// TIA Portal V19 export
ORGANIZATION_BLOCK "Main"   // OB1, FBD, ProgramCycle
TITLE = "Main Program Sweep (Cycle)"
{ S7_Optimized_Access := 'TRUE' }
// stored: SetENOAutomatically false
   VAR_INPUT
      Initial_Call : Bool;   // Initial call of this OB
      Remanence : Bool;   // =True, if remanent data are available
   END_VAR
   VAR_TEMP   // added for the SCL form of the ladder/FBD networks
      _w1 : Bool;
   END_VAR
BEGIN

REGION Network 1: Debug tags
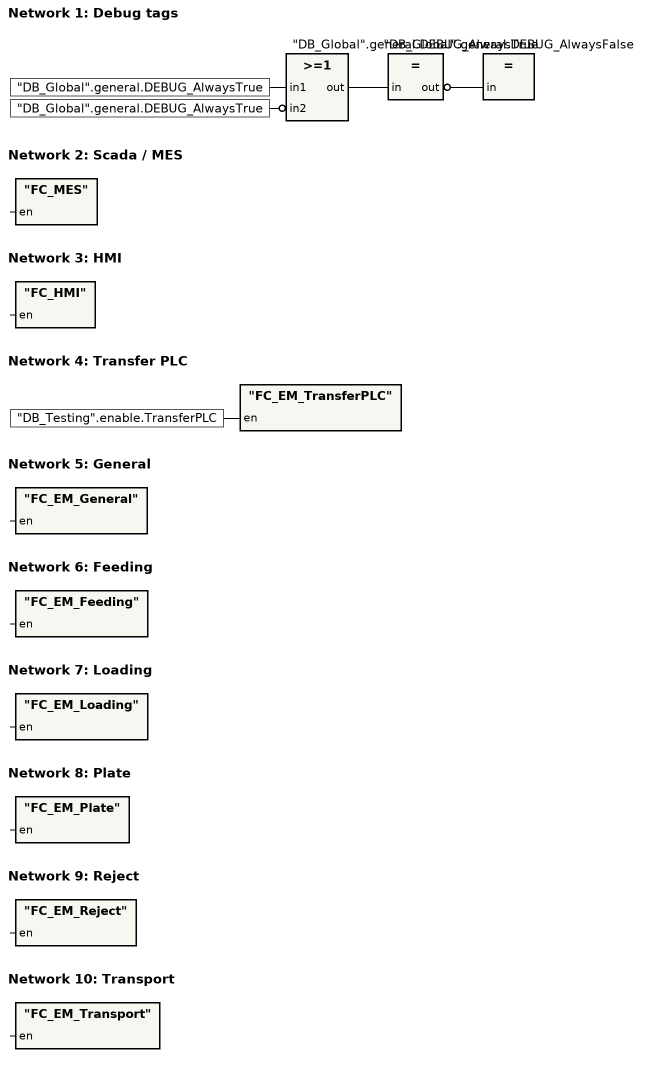
   #_w1 := "DB_Global".general.DEBUG_AlwaysTrue OR NOT "DB_Global".general.DEBUG_AlwaysTrue;
   "DB_Global".general.DEBUG_AlwaysTrue := #_w1;
   "DB_Global".general.DEBUG_AlwaysFalse := NOT #_w1;
END_REGION

REGION Network 2: Scada / MES
   "FC_MES"();
END_REGION

REGION Network 3: HMI
   "FC_HMI"();
END_REGION

REGION Network 4: Transfer PLC
   IF "DB_Testing".enable.TransferPLC THEN "FC_EM_TransferPLC"(); END_IF;
END_REGION

REGION Network 5: General
   "FC_EM_General"();
END_REGION

REGION Network 6: Feeding
   "FC_EM_Feeding"();
END_REGION

REGION Network 7: Loading
   "FC_EM_Loading"();
END_REGION

REGION Network 8: Plate
   "FC_EM_Plate"();
END_REGION

REGION Network 9: Reject
   "FC_EM_Reject"();
END_REGION

REGION Network 10: Transport
   "FC_EM_Transport"();
END_REGION
END_ORGANIZATION_BLOCK
